PROGRAM EventLoggerProgram
VAR
	bBoolean	:	BOOL;	

	eEventType		: E_EventType := E_EventType.Alarm;
	eEventSeverity	:	TcEventSeverity := TcEventSeverity.Error;
	nEventIdentity	:	UDINT := 42;
	sEventText		:	STRING(255) := 'An Error has occured';
	
	CsvPersistentEventStorage	:	FB_CsvPersistentEventStorage;
	EventLogger	:	EventLogger(CsvPersistentEventStorage);
END_VAR

IF bBoolean THEN
	EventLogger.AddEvent(eEventType, eEventSeverity, nEventIdentity, sEventText);	
	bBoolean := FALSE;
END_IF

CsvPersistentEventStorage();

END_PROGRAM

(* stored: Version 1.1.0.1, ProductVersion 3.1.4024.12
   POU EventLoggerProgram: Id {2d5e86fb-cf04-4625-9bd9-96b21eef3ebf}, SpecialFunc None *)
